FUNCTION_BLOCK EdgeDetector
VAR_INPUT
	b_StateButtonActal : BOOL;
END_VAR
VAR_OUTPUT
	s_StateEdgedetector: STRING;
END_VAR
VAR
	b_StateButtonOld : BOOL;
END_VAR

IF NOT b_StateButtonOld AND b_StateButtonActal THEN
	s_StateEdgedetector := 'risingEdge';
	
ELSIF  b_StateButtonOld AND NOT b_StateButtonActal THEN
	s_StateEdgedetector := 'falingEdge';
ELSE 
	s_StateEdgedetector := 'not Changed';
END_IF
b_StateButtonOld := b_StateButtonActal;

END_FUNCTION_BLOCK

(* stored: Version 1.1.0.1, ProductVersion 3.1.4022.12
   POU EdgeDetector: Id {b4aa9d4b-350f-4690-8998-8c8fe231252d}, SpecialFunc None *)
